// TIA Portal V20 export
DATA_BLOCK "EventsData"   // DB496
// stored: Access Published, MemoryReserve 100, Namespace Unit1
   VAR
      ResourceData { ExternalAccessible := 'False'; ExternalVisible := 'False'; ExternalWritable := 'False'} : "LPFE_typeResourceData";
      ValueEvent : Array[0..99] of "LPFE_typeValueEventData";
      TelemetryContent : Array[0..20] of "LPFE_typeTelemetryContent";
      Transaction1_Electrodes1_30 { ExternalAccessible := 'False'; ExternalVisible := 'False'; ExternalWritable := 'False'} : "LPFE_typeFlexNetData_18000";
      Transaction2_Electrodes31_60 { ExternalAccessible := 'False'; ExternalVisible := 'False'; ExternalWritable := 'False'} : "LPFE_typeFlexNetData_18000";
      Transaction3_Electrodes61_90 { ExternalAccessible := 'False'; ExternalVisible := 'False'; ExternalWritable := 'False'} : "LPFE_typeFlexNetData_18000";
      RecordGenericPayload { S7_SetPoint := 'True'} : "LPFE_typeRecordGenericPayload";
   END_VAR
BEGIN
   ResourceData.resourceInterestID := 10;
END_DATA_BLOCK
